# B&R Automation Studio project GettingStarted_MpPick (part 2)

#### Main.st
```iecst
PROGRAM _INIT

    PC_Step := PC_ENABLE_PICK_CORE;
    Gripper := FALSE;

END_PROGRAM

PROGRAM _CYCLIC

    CASE PC_Step OF

        (* Enable the PickCore *)
        PC_ENABLE_PICK_CORE:
            MpPickCore_0.Enable := TRUE;
            PC_Step := PC_WAIT_ENABLE_PICK_CORE;

        PC_WAIT_ENABLE_PICK_CORE:
            IF MpPickCore_0.Active THEN
                PC_Step := PC_ENABLE_CORE_PROCESS;

			ELSIF MpPickCore_0.Error THEN
				LastStep := PC_Step;
                PC_Step  := PC_ERROR;

			END_IF;

        PC_ENABLE_CORE_PROCESS:
            MpPickCore_0.ProcessEnable := TRUE;
            PC_Step := PC_WAIT_ENABLE_CORE_PROCESS;

        PC_WAIT_ENABLE_CORE_PROCESS:
            IF MpPickCore_0.ProcessActive THEN
                PC_Step := PC_READY_TO_START;

            ELSIF MpPickCore_0.Error THEN
				LastStep := PC_Step;
                PC_Step  := PC_ERROR;

            END_IF

        PC_READY_TO_START:
            ReadyPickCore := TRUE;

            IF CmdStart THEN
                MpPickCore_0.Parameters.OperationMode := 'ConveyorToConveyor';
			    MpPickCore_0.ProcessStart := TRUE;
                PC_Step := PC_WAIT_START_CORE_PROCESS;
            END_IF

        PC_WAIT_START_CORE_PROCESS:
			IF MpPickCore_0.ProcessRunning THEN
                PC_Step := PC_STARTED;

			ELSIF MpPickCore_0.Error THEN
				LastStep := PC_Step;
                PC_Step  := PC_ERROR;

			END_IF;

        PC_STARTED:
            (* Nothing to do here *)
            IF MpPickCore_0.Error THEN
				LastStep := PC_Step;
                PC_Step  := PC_ERROR;
			END_IF;

        PC_ERROR:
            Error := TRUE;
            ReadyPickCore := FALSE;

    END_CASE

    (* Call FBs *)
    MpPickCore_0.MpLink := ADR(gPickCore_1);
    MpPickCore_0();

END_PROGRAM
```

### Program Logical/PickAndPlace/PrgPlace

#### Types.typ
```iecst
TYPE
	PlaceStepEnum :
		(
		P_WAIT_ENABLE,
		P_ENABLE_REGISTER_FB,
		P_WAIT_ENABLE_REGISTER_FB,
		P_ENABLE_REGISTER_COMP,
		P_WAIT_ENABLE_REGISTER_COMP,
		P_ENABLE_ADD_REGISTER_FBS,
		P_WAIT_ENABLE_ADD_REGISTER_FBS,
		P_WAIT_START_PROCESS,
		P_CREATE_OBJECTS,
		P_WAIT_CREATE_OBJECTS,
		P_WAIT_REGISTER_FULL,
		P_DELAY_DELETE,
		P_DELETE_OBJECTS,
		P_WAIT_DELETE_OBJECTS,
		P_DELAY_CREATE,
		P_ERROR
		);
END_TYPE
```

#### Variables.var
```iecst
VAR
	P_Step : PlaceStepEnum;
	LastStep : PlaceStepEnum;
	Error : BOOL;
	PlaceHoldersSpacing : LREAL;
	LastPlaceHolderConveyorPosition : LREAL;
	ElapsedDistance : LREAL;
END_VAR
(*   *)
(*Functionblocks*)
VAR
	MpPickRegister_0 : MpPickRegister;
	MpPickRegCreatePlaceholder : MpPickRegCreateObject;
END_VAR
```

#### Main.st
```iecst
PROGRAM _INIT

    P_Step := P_WAIT_ENABLE;
    Error := FALSE;

    PlaceHoldersSpacing := 65.0; // distance between two consecutive place holders

END_PROGRAM

PROGRAM _CYCLIC

    CASE P_Step OF
        P_WAIT_ENABLE:
            P_Step := P_ENABLE_REGISTER_FB;

        P_ENABLE_REGISTER_FB:
            MpPickRegister_0.Enable := TRUE;
            P_Step := P_WAIT_ENABLE_REGISTER_FB;

        P_WAIT_ENABLE_REGISTER_FB:
            IF MpPickRegister_0.Active THEN
                P_Step := P_ENABLE_REGISTER_COMP;

            ELSIF MpPickRegister_0.Error THEN
                LastStep := P_Step;
                P_Step := P_ERROR;
            END_IF;

        P_ENABLE_REGISTER_COMP:
            MpPickRegister_0.RegisterEnable := TRUE;
            P_Step := P_WAIT_ENABLE_REGISTER_COMP;

        P_WAIT_ENABLE_REGISTER_COMP:
            IF MpPickRegister_0.RegisterActive THEN
                P_Step := P_ENABLE_ADD_REGISTER_FBS;

            ELSIF MpPickRegister_0.Error THEN
                LastStep := P_Step;
                P_Step := P_ERROR;
            END_IF;

        P_ENABLE_ADD_REGISTER_FBS:
            MpPickRegCreatePlaceholder.Enable := TRUE;
            MpPickRegCreatePlaceholder.Create := FALSE;
            P_Step := P_WAIT_ENABLE_ADD_REGISTER_FBS;

        P_WAIT_ENABLE_ADD_REGISTER_FBS:
            IF 	MpPickRegCreatePlaceholder.Active THEN
                P_Step := P_WAIT_START_PROCESS;

            ELSIF MpPickRegCreatePlaceholder.Error THEN
                LastStep := P_Step;
                P_Step := P_ERROR;
            END_IF;

        P_WAIT_START_PROCESS: // waits user start command and conveyor moving
            ReadyPlaceReg := TRUE;
            IF CmdStart AND ReadyToStart AND (PlaceConveyorPosition > 0) THEN
                P_Step := P_CREATE_OBJECTS;
            END_IF;

        (* We need to create positions (place holders) on place conveyor where to place picked objects *)
        P_CREATE_OBJECTS:

            ElapsedDistance := DistanceOverPeriod(PlaceConveyorPosition, LastPlaceHolderConveyorPosition, PlaceConveyorLength);

            IF (ElapsedDistance >= PlaceHoldersSpacing) THEN

                MpPickRegCreatePlaceholder.Parameters.LatchedConveyor.Position := PlaceConveyorPosition;
                MpPickRegCreatePlaceholder.Parameters.Mode := mpPICK_CREATE_SINGLEITEM_PLACEH;
                MpPickRegCreatePlaceholder.Parameters.ObjectTypeName := 'MyProduct';
                MpPickRegCreatePlaceholder.Parameters.Translation.X := 0;
                MpPickRegCreatePlaceholder.Parameters.Translation.Y := 125; // in the middle of conveyor width
                MpPickRegCreatePlaceholder.Create := TRUE;

                LastPlaceHolderConveyorPosition := MpPickRegCreatePlaceholder.Parameters.LatchedConveyor.Position;
            ELSE
                MpPickRegCreatePlaceholder.Create := FALSE;
            END_IF

        P_ERROR:
            Error := TRUE;
            ReadyPlaceReg := FALSE;

    END_CASE;

    (* FB calls *)
    MpPickRegister_0.MpLink := ADR(gPlaceRegister);
    MpPickRegister_0();

    MpPickRegCreatePlaceholder.MpLink := ADR(gPlaceRegister);
	MpPickRegCreatePlaceholder();

END_PROGRAM
```

Listed in the project but not available here: Logical/Global.typ, Logical/Global.var
